TYPE ioBundleControl :
STRUCT
	
	
END_STRUCT
END_TYPE

(* stored: Version 1.1.0.1, ProductVersion 3.1.4024.0
   DUT ioBundleControl: Id {45aca38f-7357-436a-a68f-baff3d088c5e} *)
